(*
Nazwa:			E_CatchStationState
Opis:			Stany chwytaka
Wersja:			v0.2
Data:			2018-10-18
Autor:			TW
Urzadzenia:		
Konfiguracja:	
Info:
-nowy stan
*)

TYPE E_CatchStationState :
(
	eDisabled:=0,  			//Wyłączona
	eError:=1,				//Błąd
	eManualMovement:=2,		//Tryb serwisowy
	eHoming:=4,				//Bazowanie
	eHomingDone:=5,			//Koniec bazowania
	eReady:=6,				//Gotowość
	eCatching:=7, 			//Chwytanie
	eCatched:=8,  			//Chwycono
	ePreparingToDisable:=9, (*NOWY*) //Przygotowanie do wyłączenia
	eNotCatched:=10       //NIe złapało
):=eDisabled;
END_TYPE

(* stored: Version 1.1.0.1, ProductVersion 3.1.4026.13, FileIdentifier bd3657e3d47ccdc489cdc2e5b8e060399c404da5, FileSignature 5fefca502ad1e5af98ece6c1335e950f73dd4f1ee1eed3100d079b845723e8413c3fcfad3b1a2c9fa27998757ccaef04abf2c8f9e4d3a5d82ae2068e9d30bb1ba41b587b1c839db346df08d0875620fbc6a4fcc82c2fd0b79e667988ce1b05df647a34fde6991ec3fdc44a5e6ab6f1e2eaca4246f58e3359c2f5461c379b309559ab035b79c30ea3c68c1507b68a309436b70e72bfaf12bce4a816a7c57be9a57020a8ff963513729d3010753251dc99dfa8d1872b3253120e9f0039ec534a289f1bd6ef610e3de698eaa14109d9db5059f87c59361849fe8e9822e7e97c90b1173215f15a6d8904971862c466faf1fc1ed82b2767e11d46c0e558f7c4338b66
   DUT E_CatchStationState: Id {711d07ca-9c02-4274-8f95-b6fffc59dcc4} *)
